INTERFACE itfContinuousAxisCommand EXTENDS itfAxisCommand

PROPERTY InVelocity : BOOL
GET
END_GET
END_PROPERTY

END_INTERFACE

(* stored: Version 1.1.0.1, ProductVersion 3.1.4024.12
   Itf itfContinuousAxisCommand: Id {f57eb851-23f6-4e4a-8fc3-1f699263815c}
   Property InVelocity: Id {6763be39-fe04-48bc-98bd-d8144ddf71ec}
   Get Get: Id {6b7b0bb7-0ddd-4dc5-9076-5b55c8f3d2f9} *)
